FUNCTION_BLOCK FB_AxisControl
VAR_INPUT
	xEnable: BOOL;
	xZero: BOOL;
	xMoveR: BOOL;
	xMoveA: BOOL;
	xMoveV: BOOL;
	xPositiveDirection: BOOL;
	fDistance: LREAL;
	fPosition: LREAL;
	fVelocity: LREAL;
	xStop: BOOL;
	xHome: BOOL;
	xHomeFlag: BOOL;
	xHalt: BOOL;
	xTimerInput: BOOL;
	timerPT: TIME;
	HomePosition: LREAL;
	fAxisAcceleration: LREAL;
	fAxisDeceleration: LREAL;
	fAxisJerk: LREAL;
	MasterAxis: AXIS_REF;
	GearIn: BOOL;
	Gear_out: BOOL;
	GearRatio: LREAL;
	EnableSoE_ReadPosition: BOOL;
	EnableSoE_ReadTorque: BOOL;
	EnableSoE_ReadFollowingError: BOOL;
	fHomeOffset: LREAL;
END_VAR
VAR_OUTPUT
	gear_out_busy	:BOOL;
	fActualPosition: LREAL;
	fActualVelocity: LREAL;
	fActModuloPos: LREAL;
	fActPosition: DINT;
	fActFollowingError: DINT;
	fActualTorque: INT;
	xEnabled: BOOL;
	xMoveComplete: BOOL;
	xInPosition: BOOL;
	xAtSpeed: BOOL;
	xStopped: BOOL;
	xHomed: BOOL;
	xHalted: BOOL;
	errorID: UDINT;
	xAxisHomed: BOOL;
	xZeroed: BOOL;
	timerET: TIME;
	timerQOutput: BOOL;
	InGear: BOOL;
	xServoError: BOOL;
	iErrorID: UDINT;
END_VAR
VAR
	mcPower: MC_Power;
	mcReset: MC_Reset;
	mcMoveRelative: MC_MoveRelative;
	mcSetPosition: MC_SetPosition;
	mcMoveAbsolute: MC_MoveAbsolute;
	mcReadStatus: MC_ReadStatus;
	mcMoveVelocity: MC_MoveVelocity;
	mcStop: MC_Stop;
	mcHome: MC_Home;
	mcHalt: MC_Halt;
	timerOn: TON;

	mcGearInDyn: MC_GearInDyn;
	mcGearOut: MC_GearOut;
	
	EnReadPosition: BOOL;
	EnReadTorque: BOOL;
	EnReadFollowingError: BOOL;
	
END_VAR
VAR_IN_OUT
	Axis: AXIS_REF;
	//MasterAxis : AXIS_REF;
END_VAR

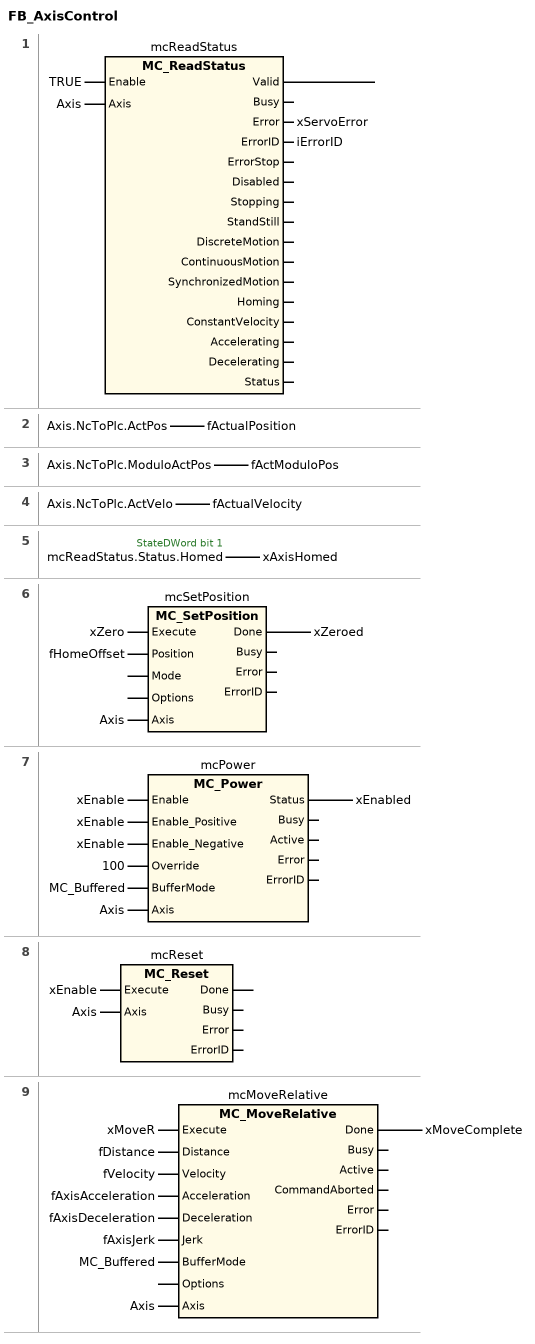
// NETWORK 1
mcReadStatus(Enable := TRUE, Axis := Axis, Error => xServoError, ErrorID => iErrorID); // MC_ReadStatus

// NETWORK 2
fActualPosition := Axis.NcToPlc.ActPos;

// NETWORK 3
fActModuloPos := Axis.NcToPlc.ModuloActPos;

// NETWORK 4
fActualVelocity := Axis.NcToPlc.ActVelo;

// NETWORK 5
//   mcReadStatus.Status.Homed: StateDWord bit 1
xAxisHomed := mcReadStatus.Status.Homed;

// NETWORK 6
mcSetPosition(Execute := xZero, Position := fHomeOffset, Axis := Axis); // MC_SetPosition
xZeroed := mcSetPosition.Done;

// NETWORK 7
mcPower(
    Enable := xEnable,
    Enable_Positive := xEnable,
    Enable_Negative := xEnable,
    Override := 100,
    BufferMode := MC_Buffered,
    Axis := Axis); // MC_Power
xEnabled := mcPower.Status;

// NETWORK 8
mcReset(Execute := xEnable, Axis := Axis); // MC_Reset

// NETWORK 9
mcMoveRelative(
    Execute := xMoveR,
    Distance := fDistance,
    Velocity := fVelocity,
    Acceleration := fAxisAcceleration,
    Deceleration := fAxisDeceleration,
    Jerk := fAxisJerk,
    BufferMode := MC_Buffered,
    Axis := Axis); // MC_MoveRelative
xMoveComplete := mcMoveRelative.Done;

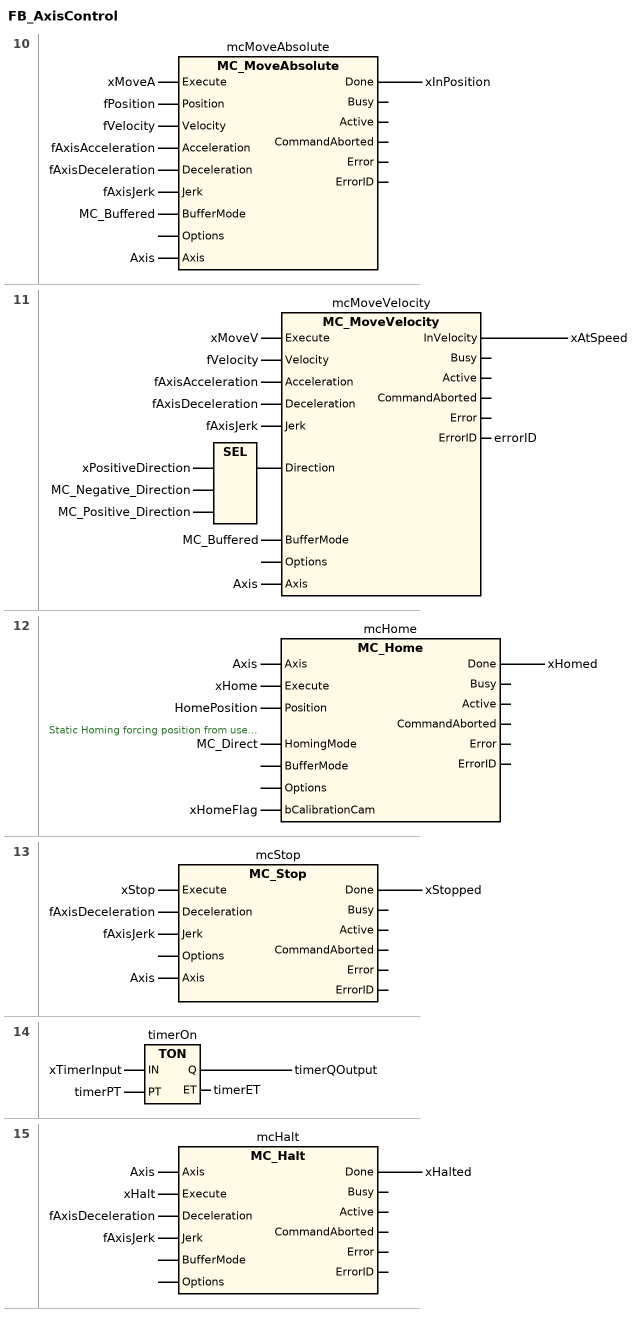
// NETWORK 10
mcMoveAbsolute(
    Execute := xMoveA,
    Position := fPosition,
    Velocity := fVelocity,
    Acceleration := fAxisAcceleration,
    Deceleration := fAxisDeceleration,
    Jerk := fAxisJerk,
    BufferMode := MC_Buffered,
    Axis := Axis); // MC_MoveAbsolute
xInPosition := mcMoveAbsolute.Done;

// NETWORK 11
mcMoveVelocity(
    Execute := xMoveV,
    Velocity := fVelocity,
    Acceleration := fAxisAcceleration,
    Deceleration := fAxisDeceleration,
    Jerk := fAxisJerk,
    Direction := SEL(xPositiveDirection, MC_Negative_Direction, MC_Positive_Direction),
    BufferMode := MC_Buffered,
    Axis := Axis,
    ErrorID => errorID); // MC_MoveVelocity
xAtSpeed := mcMoveVelocity.InVelocity;

// NETWORK 12
//   MC_Direct: Static Homing forcing position from user reference
mcHome(
    Axis := Axis,
    Execute := xHome,
    Position := HomePosition,
    HomingMode := MC_Direct,
    bCalibrationCam := xHomeFlag); // MC_Home
xHomed := mcHome.Done;

// NETWORK 13
mcStop(Execute := xStop, Deceleration := fAxisDeceleration, Jerk := fAxisJerk, Axis := Axis); // MC_Stop
xStopped := mcStop.Done;

// NETWORK 14
timerOn(IN := xTimerInput, PT := timerPT, ET => timerET); // TON
timerQOutput := timerOn.Q;

// NETWORK 15
mcHalt(Axis := Axis, Execute := xHalt, Deceleration := fAxisDeceleration, Jerk := fAxisJerk); // MC_Halt
xHalted := mcHalt.Done;

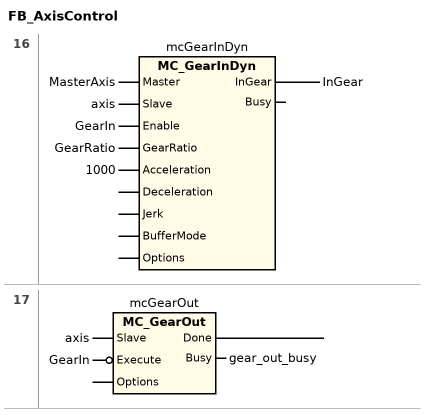
// NETWORK 16
mcGearInDyn(
    Master := MasterAxis,
    Slave := axis,
    Enable := GearIn,
    GearRatio := GearRatio,
    Acceleration := 1000); // MC_GearInDyn
InGear := mcGearInDyn.InGear;

// NETWORK 17
mcGearOut(Slave := axis, Execute := NOT GearIn, Busy => gear_out_busy); // MC_GearOut

END_FUNCTION_BLOCK

(* stored: Version 1.1.0.1, ProductVersion 3.1.4020.12
   POU FB_AxisControl: Id {55212095-de5e-4714-a460-98605f7fc17e}, SpecialFunc None *)
